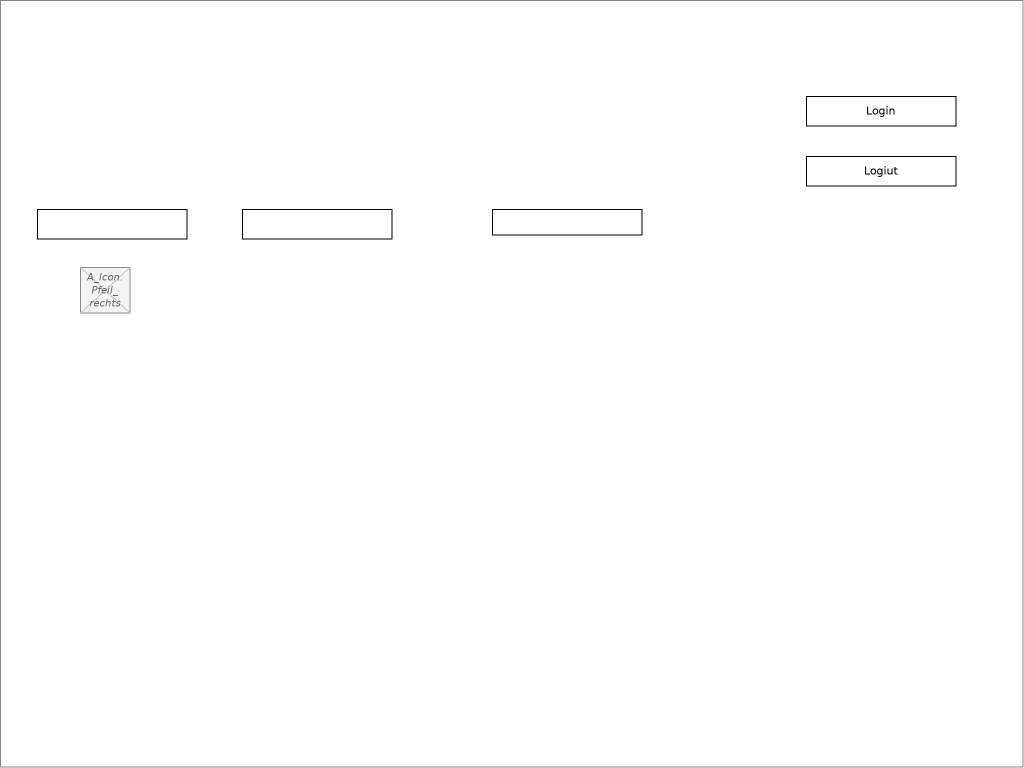
VISUALIZATION Test_Login  // 1024x768
VAR_IN_OUT
	FB_AI_8:AI_8;
END_VAR
    Rectangle (37,209 150x30)
        OnMouseClick: change screen: Home
    Rectangle (242,209 150x30)
        OnMouseClick: change screen: Home
    Rectangle (492,209 150x26)
    Rectangle (806,96 150x30), "Login"
        OnMouseClick: VisuUserMgmt Type=Login
    Rectangle (806,156 150x30), "Logiut"
        OnMouseClick: VisuUserMgmt Type=Logout
    Image (80,267 50x46), image: A_Icon.Pfeil_rechts
        OnMouseClick: execute { Visu.i_Frame_VD_Index:=4; }
END_VISUALIZATION

(* stored: Version 1.1.0.1, ProductVersion 3.1.4022.6
   Visu Test_Login: Id {47986cee-6727-4c50-9eb6-91cce4a4b8b2} *)
